// TIA Portal V17 export
// export: Created 2023-04-07T09:07:26.8247712Z, ExportSetting WithDefaults, DisplayName Totally Integrated Automation Portal, DisplayVersion V17 Update 4, DisplayName TIA Portal Openness, DisplayVersion V17 Update 4, DisplayName TIA Portal Version Control Interface, DisplayVersion V17, DisplayName STEP 7 Professional, DisplayVersion V17 Update 4, DisplayName STEP 7 Safety, DisplayVersion V17, DisplayName WinCC Professional, DisplayVersion V17 Update 4
TYPE "RW_PE"
// stored: IsFailsafeCompliant false
   STRUCT
      iUserPswIns : Int;
      iModePctrlCmd : Int;
      iModeQctrlCmd : Int;
      rPacRef : Real;
      rQacRef : Real;
      xStartCmd : Bool;
      xGeneral_SelectorEnable : Bool;
      xDC_SelectorEnable : Bool;
      xDC_VirtualSelector : Bool;
      xAC_SelectorEnable : Bool;
      xAC_VirtualSelector : Bool;
      xStopCmd : Bool;
      xClearFltCmd : Bool;
      xEmeStopCmd : Bool;
      xEnableCmd : Bool;
      wBankDcEnbCmd : Word;
      iWatchDog : Int;
      xMVskid_comm : Bool;   // Register 41880 | 0 = communications enabled
      uiMVskid_CB : UInt;   // Register 41881 | 1=open; 2=closed; 0=idle;
   END_STRUCT;
END_TYPE
